// TIA Portal V20 export
TYPE "LER_typeEmRelation"
// stored: Access Published
   STRUCT
      UserDefine : "LER_typeUserDefine";   // User Define
      softCam : Array[0..11] of "LER_typeSoftCamRelation";   // Axis Position Check
      cmStatus : "LER_typeCmStatus";   // Control Modules Status
      sequence : Array[0..19] of "LER_typeSequenceRelation";   // Em Sequence
   END_STRUCT;
END_TYPE
